// TIA Portal V18 export
DATA_BLOCK "SS1_A8_16DI_16DO_DO_Vars"   // DB11082
{ S7_Optimized_Access := 'FALSE' }
VERSION : 0.1
// stored: AutoNumber false, DBAccessibleFromOPCUA true, IsOnlyStoredInLoadMemory false, IsWriteProtectedInAS false
   VAR
      DO1 { S7_SetPoint := 'True'} : "UDT_DOadv";
      DO2 { S7_SetPoint := 'True'} : "UDT_DOadv";
      DO3 { S7_SetPoint := 'True'} : "UDT_DOadv";
      DO4 { S7_SetPoint := 'True'} : "UDT_DOadv";
      DO5 { S7_SetPoint := 'True'} : "UDT_DOadv";
      DO6 { S7_SetPoint := 'True'} : "UDT_DOadv";
      DO7 { S7_SetPoint := 'True'} : "UDT_DOadv";
      DO8 { S7_SetPoint := 'True'} : "UDT_DOadv";
      DO9 { S7_SetPoint := 'True'} : "UDT_DOadv";
      DO10 { S7_SetPoint := 'True'} : "UDT_DOadv";
      DO11 { S7_SetPoint := 'True'} : "UDT_DOadv";
      DO12 { S7_SetPoint := 'True'} : "UDT_DOadv";
      DO13 { S7_SetPoint := 'True'} : "UDT_DOadv";
      DO14 { S7_SetPoint := 'True'} : "UDT_DOadv";
      DO15 { S7_SetPoint := 'True'} : "UDT_DOadv";
      DO16 { S7_SetPoint := 'True'} : "UDT_DOadv";
   END_VAR
BEGIN
   DO1.iFuncSystemID := 1;
   DO1.iFuncVar := 4;
   DO2.iFuncSystemID := 1;
   DO3.iFuncSystemID := 1;
   DO4.iFuncSystemID := 1;
   DO5.iFuncSystemID := 1;
   DO6.cMOA := 1;
   DO7.iFuncSystemID := 3;
   DO7.iFuncVar := 1;
   DO7.cMOA := 1;
   DO8.iFuncSystemID := 3;
   DO9.iFuncSystemID := 3;
   DO9.iFuncVar := 3;
   DO13.iFuncSystemID := 10;
   DO13.iFuncVar := 1;
   DO14.iFuncSystemID := 10;
   DO14.iFuncVar := 2;
   DO15.iFuncSystemID := 10;
   DO15.iFuncVar := 3;
   DO16.iFuncSystemID := 10;
   DO16.iFuncVar := 4;
END_DATA_BLOCK
